ABB RobotStudio station: Lab5.rsstnx

Station Lab5 (saved by RobotStudio 24.3.10885.0)
Layout (positions relative to the parent item):
